TYPE HoursStruct :
STRUCT
END_STRUCT
END_TYPE

(* stored: Version 1.1.0.1, ProductVersion 3.1.4024.4
   DUT HoursStruct: Id {c6aa12e2-a7c8-45ca-95ee-49a689f30a49} *)
